// TIA Portal project "Soru3" (V15)

(* hardware
DEVICE "S7-1200 station_1"  S7-1200 Station
   slot 0: "Rack_0"  S7-1200 Rack  Rack  V1.0
   slot 1: "PLC_1"  CPU 1214C DC/DC/DC  6ES7 214-1AG40-0XB0  V4.2
*)

// ===== PLC "PLC_1"  CPU 1214C DC/DC/DC =====

VAR_GLOBAL   // PLC tag table "Default tag table"
   "Başlat" AT %I0.1 : Bool;
   "Dur" AT %I0.0 : Bool;
   "Motor_Yıldız" AT %Q0.0 : Bool;
   "Motor_Ucgen" AT %Q0.1 : Bool;
   "Motor_D_Fren" AT %Q0.2 : Bool;
END_VAR

// folder: System blocks/Program resources

DATA_BLOCK "IEC_Timer_0_DB"   // DB1
{ S7_Optimized_Access := 'TRUE' }
AUTHOR : Simatic
FAMILY : IEC
NAME : IEC_TMR
VERSION : 1.0
// stored: InstanceOfName IEC_TIMER
"IEC_TIMER"
BEGIN
END_DATA_BLOCK

// folder: (top level)

ORGANIZATION_BLOCK "Main"   // OB1, LAD, ProgramCycle
TITLE = "Main Program Sweep (Cycle)"
{ S7_Optimized_Access := 'TRUE' }
VERSION : 0.1
   VAR_INPUT
      Initial_Call : Bool;   // Initial call of this OB
      Remanence : Bool;   // =True, if remanent data are available
   END_VAR
BEGIN

REGION Network 1: 10 saniyeden düşükte yıldız, 10saniye sonra üçigen
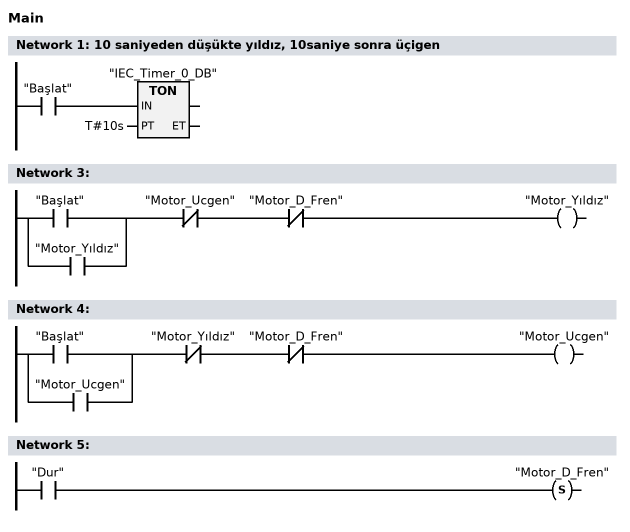
   "IEC_Timer_0_DB".TON(IN := "Başlat", PT := T#10s);
END_REGION

REGION Network 3
   RUNG wire#powerrail
      Contact( "Başlat" )
      wire#w1
      I_Contact( "Motor_Ucgen" )
      I_Contact( "Motor_D_Fren" )
      Coil( "Motor_Yıldız" )
   END_RUNG
   RUNG wire#powerrail
      Contact( "Motor_Yıldız" )
   END_RUNG wire#w1
   // the same network as SCL:
   "Motor_Yıldız" := ("Başlat" OR "Motor_Yıldız") AND NOT "Motor_Ucgen" AND NOT "Motor_D_Fren";
END_REGION

REGION Network 4
   RUNG wire#powerrail
      Contact( "Başlat" )
      wire#w1
      I_Contact( "Motor_Yıldız" )
      I_Contact( "Motor_D_Fren" )
      Coil( "Motor_Ucgen" )
   END_RUNG
   RUNG wire#powerrail
      Contact( "Motor_Ucgen" )
   END_RUNG wire#w1
   // the same network as SCL:
   "Motor_Ucgen" := ("Başlat" OR "Motor_Ucgen") AND NOT "Motor_Yıldız" AND NOT "Motor_D_Fren";
END_REGION

REGION Network 5
   RUNG wire#powerrail
      Contact( "Dur" )
      S_Coil( "Motor_D_Fren" )
   END_RUNG
   // the same network as SCL:
   IF "Dur" THEN "Motor_D_Fren" := TRUE; END_IF;
END_REGION
END_ORGANIZATION_BLOCK